  MoveL 1298 to (-37.11, 208.63, 290) mm, rotated rx -90 ry -25 rz 8.11 deg; joints [2.992, -45.692, 98.056, 40.659, -108.852, -6.827, -2568.107]
  MoveL 1299 to (-37.11, 208.63, 290) mm, rotated rx -90 ry -25 rz 8.11 deg; joints [2.992, -45.692, 98.056, 40.659, -108.852, -6.827, -2568.107]
  Set speed (60.0 mm/s)
  MoveL 1300 to (-43.85, 188.95, 290) mm, rotated rx -90 ry -25 rz 14.31 deg; joints [2.992, -46.574, 97.966, 40.447, -108.114, -7.494, -2574.314]
  Set speed (1000.0 mm/s)
  MoveL 1301 to (-43.85, 188.95, 290) mm, rotated rx -90 ry -25 rz 14.31 deg; joints [2.992, -46.574, 97.966, 40.447, -108.114, -7.494, -2574.314]
  Set speed (1000.0 mm/s)
  MoveL 1302 to (20.49, 309.71, 0) mm, rotated rx -90 ry -25 rz -148.94 deg; joints [-7.468, -50.346, 106.416, 34.531, -108.048, 0.653, -2411.057]
  MoveL 1303 to (20.49, 309.71, 0) mm, rotated rx -90 ry -25 rz -148.94 deg; joints [-7.468, -50.346, 106.416, 34.531, -108.048, 0.653, -2411.057]
  Set speed (60.0 mm/s)
  MoveL 1304 to (20.57, 330.51, 0) mm, rotated rx -90 ry -25 rz -144.34 deg; joints [-7.468, -51.311, 106.31, 34.338, -107.164, 0.017, -2415.665]
  Set speed (1000.0 mm/s)
  MoveL 1305 to (20.57, 330.51, 0) mm, rotated rx -90 ry -25 rz -144.34 deg; joints [-7.468, -51.311, 106.31, 34.338, -107.164, 0.017, -2415.665]
  Set speed (1000.0 mm/s)
  MoveL 1306 to (20.49, 309.71, 0) mm, rotated rx -90 ry -25 rz -148.94 deg; joints [-7.468, -50.346, 106.416, 34.531, -108.048, 0.653, -2411.057]
  MoveL 1307 to (20.49, 309.71, 0) mm, rotated rx -90 ry -25 rz -148.94 deg; joints [-7.468, -50.346, 106.416, 34.531, -108.048, 0.653, -2411.057]
  Set speed (60.0 mm/s)
  MoveL 1308 to (16.38, 311.06, 10) mm, rotated rx -90 ry -25 rz -145.01 deg; joints [-7.088, -50.246, 106.214, 34.77, -108.084, 0.408, -2414.985]
  MoveL 1309 to (11.76, 312.2, 20) mm, rotated rx -90 ry -25 rz -140.7 deg; joints [-6.709, -50.143, 106.006, 35.007, -108.12, 0.162, -2419.296]
  MoveL 1310 to (6.67, 313.01, 30) mm, rotated rx -90 ry -25 rz -136.04 deg; joints [-6.332, -50.036, 105.793, 35.242, -108.155, -0.085, -2423.955]
  MoveL 1311 to (1.18, 313.37, 40) mm, rotated rx -90 ry -25 rz -131.07 deg; joints [-5.956, -49.924, 105.573, 35.476, -108.19, -0.333, -2428.933]
  MoveL 1312 to (-4.64, 313.2, 50) mm, rotated rx -90 ry -25 rz -125.8 deg; joints [-5.581, -49.807, 105.347, 35.708, -108.224, -0.581, -2434.198]
  MoveL 1313 to (-10.69, 312.41, 60) mm, rotated rx -90 ry -25 rz -120.28 deg; joints [-5.207, -49.684, 105.115, 35.938, -108.259, -0.83, -2439.72]
  MoveL 1314 to (-16.86, 310.92, 70) mm, rotated rx -90 ry -25 rz -114.53 deg; joints [-4.834, -49.556, 104.876, 36.166, -108.295, -1.078, -2445.47]
  MoveL 1315 to (-23.03, 308.7, 80) mm, rotated rx -90 ry -25 rz -108.58 deg; joints [-4.463, -49.423, 104.632, 36.393, -108.331, -1.327, -2451.421]
  MoveL 1316 to (-29.06, 305.72, 90) mm, rotated rx -90 ry -25 rz -102.46 deg; joints [-4.093, -49.283, 104.382, 36.619, -108.368, -1.575, -2457.545]
  MoveL 1317 to (-34.83, 302, 100) mm, rotated rx -90 ry -25 rz -96.19 deg; joints [-3.725, -49.138, 104.126, 36.842, -108.405, -1.823, -2463.814]
  MoveL 1318 to (-40.19, 297.56, 110) mm, rotated rx -90 ry -25 rz -89.8 deg; joints [-3.358, -48.988, 103.864, 37.064, -108.442, -2.072, -2470.201]
  MoveL 1319 to (-45.04, 292.47, 120) mm, rotated rx -90 ry -25 rz -83.32 deg; joints [-2.992, -48.832, 103.595, 37.285, -108.48, -2.32, -2476.68]
  MoveL 1320 to (-49.26, 286.82, 130) mm, rotated rx -90 ry -25 rz -76.78 deg; joints [-2.628, -48.671, 103.321, 37.503, -108.518, -2.569, -2483.221]
  MoveL 1321 to (-52.77, 280.72, 140) mm, rotated rx -90 ry -25 rz -70.2 deg; joints [-2.265, -48.505, 103.04, 37.719, -108.556, -2.819, -2489.796]
  MoveL 1322 to (-55.51, 274.28, 150) mm, rotated rx -90 ry -25 rz -63.63 deg; joints [-1.904, -48.334, 102.753, 37.934, -108.592, -3.069, -2496.375]
  MoveL 1323 to (-57.45, 267.65, 160) mm, rotated rx -90 ry -25 rz -57.07 deg; joints [-1.544, -48.16, 102.46, 38.146, -108.628, -3.32, -2502.926]
  MoveL 1324 to (-58.59, 260.95, 170) mm, rotated rx -90 ry -25 rz -50.58 deg; joints [-1.185, -47.982, 102.161, 38.356, -108.662, -3.573, -2509.416]
  MoveL 1325 to (-58.95, 254.32, 180) mm, rotated rx -90 ry -25 rz -44.19 deg; joints [-0.828, -47.801, 101.855, 38.563, -108.694, -3.828, -2515.809]
  MoveL 1326 to (-58.59, 247.88, 190) mm, rotated rx -90 ry -25 rz -37.93 deg; joints [-0.473, -47.618, 101.543, 38.768, -108.724, -4.086, -2522.068]
  MoveL 1327 to (-57.57, 241.75, 200) mm, rotated rx -90 ry -25 rz -31.84 deg; joints [-0.119, -47.432, 101.224, 38.971, -108.752, -4.345, -2528.155]
  MoveL 1328 to (-56, 236.01, 210) mm, rotated rx -90 ry -25 rz -25.97 deg; joints [0.233, -47.244, 100.899, 39.17, -108.776, -4.608, -2534.028]
  MoveL 1329 to (-53.98, 230.73, 220) mm, rotated rx -90 ry -25 rz -20.35 deg; joints [0.584, -47.055, 100.567, 39.367, -108.797, -4.873, -2539.646]
  MoveL 1330 to (-51.62, 225.97, 230) mm, rotated rx -90 ry -25 rz -15.04 deg; joints [0.933, -46.864, 100.228, 39.56, -108.815, -5.142, -2544.964]
  MoveL 1331 to (-49.06, 221.75, 240) mm, rotated rx -90 ry -25 rz -10.06 deg; joints [1.28, -46.672, 99.883, 39.751, -108.83, -5.414, -2549.94]
  MoveL 1332 to (-46.4, 218.08, 250) mm, rotated rx -90 ry -25 rz -5.47 deg; joints [1.626, -46.479, 99.531, 39.939, -108.841, -5.69, -2554.527]
  MoveL 1333 to (-43.78, 214.95, 260) mm, rotated rx -90 ry -25 rz -1.32 deg; joints [1.97, -46.284, 99.173, 40.123, -108.849, -5.969, -2558.681]
  MoveL 1334 to (-41.29, 212.35, 270) mm, rotated rx -90 ry -25 rz 2.36 deg; joints [2.312, -46.089, 98.807, 40.305, -108.853, -6.252, -2562.358]
  MoveL 1335 to (-39.03, 210.26, 280) mm, rotated rx -90 ry -25 rz 5.51 deg; joints [2.653, -45.891, 98.435, 40.483, -108.854, -6.538, -2565.515]
  MoveL 1336 to (-37.11, 208.63, 290) mm, rotated rx -90 ry -25 rz 8.11 deg; joints [2.992, -45.692, 98.056, 40.659, -108.852, -6.827, -2568.107]
  Set speed (1000.0 mm/s)
  MoveL 1337 to (-37.11, 208.63, 290) mm, rotated rx -90 ry -25 rz 8.11 deg; joints [2.992, -45.692, 98.056, 40.659, -108.852, -6.827, -2568.107]
  Set speed (1000.0 mm/s)
  MoveL 1338 to (-43.85, 188.95, 290) mm, rotated rx -90 ry -25 rz 14.31 deg; joints [2.992, -46.574, 97.966, 40.447, -108.114, -7.494, -2574.314]
  MoveL 1339 to (-43.85, 188.95, 290) mm, rotated rx -90 ry -25 rz 14.31 deg; joints [2.992, -46.574, 97.966, 40.447, -108.114, -7.494, -2574.314]
  Set speed (60.0 mm/s)
  MoveL 1340 to (-46.6, 190.89, 280) mm, rotated rx -90 ry -25 rz 11.75 deg; joints [2.653, -46.775, 98.344, 40.272, -108.112, -7.203, -2571.748]
  MoveL 1341 to (-49.86, 193.4, 270) mm, rotated rx -90 ry -25 rz 8.62 deg; joints [2.312, -46.974, 98.716, 40.094, -108.107, -6.916, -2568.621]
  MoveL 1342 to (-53.49, 196.56, 260) mm, rotated rx -90 ry -25 rz 4.97 deg; joints [1.97, -47.172, 99.081, 39.913, -108.099, -6.633, -2564.974]
  MoveL 1343 to (-57.36, 200.4, 250) mm, rotated rx -90 ry -25 rz 0.85 deg; joints [1.626, -47.368, 99.44, 39.729, -108.088, -6.352, -2560.848]
  MoveL 1344 to (-61.34, 204.96, 240) mm, rotated rx -90 ry -25 rz -3.71 deg; joints [1.28, -47.563, 99.791, 39.542, -108.074, -6.075, -2556.286]
  MoveL 1345 to (-65.27, 210.27, 230) mm, rotated rx -90 ry -25 rz -8.67 deg; joints [0.933, -47.757, 100.136, 39.352, -108.055, -5.802, -2551.328]
  MoveL 1346 to (-68.98, 216.33, 220) mm, rotated rx -90 ry -25 rz -13.98 deg; joints [0.584, -47.949, 100.474, 39.159, -108.034, -5.532, -2546.018]
  MoveL 1347 to (-72.31, 223.11, 210) mm, rotated rx -90 ry -25 rz -19.6 deg; joints [0.233, -48.14, 100.805, 38.963, -108.008, -5.265, -2540.399]
  MoveL 1348 to (-75.1, 230.56, 200) mm, rotated rx -90 ry -25 rz -25.49 deg; joints [-0.119, -48.329, 101.13, 38.764, -107.98, -5.001, -2534.511]
  MoveL 1349 to (-77.2, 238.6, 190) mm, rotated rx -90 ry -25 rz -31.6 deg; joints [-0.473, -48.517, 101.448, 38.563, -107.948, -4.74, -2528.397]
  MoveL 1350 to (-78.47, 247.13, 180) mm, rotated rx -90 ry -25 rz -37.9 deg; joints [-0.828, -48.703, 101.76, 38.358, -107.914, -4.481, -2522.096]
  MoveL 1351 to (-78.79, 256, 170) mm, rotated rx -90 ry -25 rz -44.35 deg; joints [-1.185, -48.886, 102.065, 38.152, -107.877, -4.226, -2515.648]
  MoveL 1352 to (-78.09, 265.05, 160) mm, rotated rx -90 ry -25 rz -50.91 deg; joints [-1.544, -49.066, 102.363, 37.942, -107.838, -3.972, -2509.09]
  MoveL 1353 to (-76.31, 274.12, 150) mm, rotated rx -90 ry -25 rz -57.54 deg; joints [-1.904, -49.244, 102.656, 37.731, -107.797, -3.719, -2502.46]
  MoveL 1354 to (-73.44, 283.02, 140) mm, rotated rx -90 ry -25 rz -64.21 deg; joints [-2.265, -49.417, 102.942, 37.517, -107.754, -3.468, -2495.79]
  MoveL 1355 to (-69.5, 291.57, 130) mm, rotated rx -90 ry -25 rz -70.88 deg; joints [-2.628, -49.587, 103.221, 37.301, -107.711, -3.218, -2489.115]
  MoveL 1356 to (-64.57, 299.61, 120) mm, rotated rx -90 ry -25 rz -77.53 deg; joints [-2.992, -49.751, 103.495, 37.083, -107.667, -2.969, -2482.468]
  MoveL 1357 to (-58.74, 306.97, 110) mm, rotated rx -90 ry -25 rz -84.12 deg; joints [-3.358, -49.911, 103.762, 36.864, -107.624, -2.72, -2475.878]
  MoveL 1358 to (-52.14, 313.53, 100) mm, rotated rx -90 ry -25 rz -90.62 deg; joints [-3.725, -50.066, 104.024, 36.642, -107.58, -2.471, -2469.376]
  MoveL 1359 to (-44.91, 319.19, 90) mm, rotated rx -90 ry -25 rz -97.01 deg; joints [-4.093, -50.215, 104.279, 36.419, -107.536, -2.222, -2462.991]
  MoveL 1360 to (-37.24, 323.88, 80) mm, rotated rx -90 ry -25 rz -103.25 deg; joints [-4.463, -50.358, 104.529, 36.195, -107.494, -1.973, -2456.752]
  MoveL 1361 to (-29.3, 327.59, 70) mm, rotated rx -90 ry -25 rz -109.31 deg; joints [-4.834, -50.496, 104.772, 35.968, -107.451, -1.724, -2450.689]
  MoveL 1362 to (-21.27, 330.31, 60) mm, rotated rx -90 ry -25 rz -115.17 deg; joints [-5.207, -50.628, 105.01, 35.74, -107.41, -1.474, -2444.831]
  MoveL 1363 to (-13.31, 332.11, 50) mm, rotated rx -90 ry -25 rz -120.79 deg; joints [-5.581, -50.755, 105.242, 35.511, -107.369, -1.225, -2439.206]
  MoveL 1364 to (-5.58, 333.04, 40) mm, rotated rx -90 ry -25 rz -126.15 deg; joints [-5.956, -50.876, 105.467, 35.28, -107.328, -0.976, -2433.845]
  MoveL 1365 to (1.77, 333.22, 30) mm, rotated rx -90 ry -25 rz -131.22 deg; joints [-6.332, -50.991, 105.687, 35.047, -107.287, -0.727, -2428.779]
  MoveL 1366 to (8.64, 332.76, 20) mm, rotated rx -90 ry -25 rz -135.96 deg; joints [-6.709, -51.103, 105.901, 34.813, -107.247, -0.478, -2424.039]
  MoveL 1367 to (14.93, 331.81, 10) mm, rotated rx -90 ry -25 rz -140.34 deg; joints [-7.088, -51.209, 106.109, 34.576, -107.206, -0.23, -2419.656]
  MoveL 1368 to (20.57, 330.51, 0) mm, rotated rx -90 ry -25 rz -144.34 deg; joints [-7.468, -51.311, 106.31, 34.338, -107.164, 0.017, -2415.665]
  Set speed (1000.0 mm/s)
  MoveL 1369 to (20.57, 330.51, 0) mm, rotated rx -90 ry -25 rz -144.34 deg; joints [-7.468, -51.311, 106.31, 34.338, -107.164, 0.017, -2415.665]
  Set speed (1000.0 mm/s)
  MoveL 1370 to (-43.85, 188.95, 290) mm, rotated rx -90 ry -25 rz 14.31 deg; joints [2.992, -46.574, 97.966, 40.447, -108.114, -7.494, -2574.314]
  MoveL 1371 to (-43.85, 188.95, 290) mm, rotated rx -90 ry -25 rz 14.31 deg; joints [2.992, -46.574, 97.966, 40.447, -108.114, -7.494, -2574.314]
  Set speed (60.0 mm/s)
  MoveL 1372 to (-28.22, 202.67, 290) mm, rotated rx -90 ry -25 rz 19.2 deg; joints [2.992, -45.67, 98.058, 40.664, -108.87, -6.811, -2579.196]
  Set speed (1000.0 mm/s)
  MoveL 1373 to (-28.22, 202.67, 290) mm, rotated rx -90 ry -25 rz 19.2 deg; joints [2.992, -45.67, 98.058, 40.664, -108.87, -6.811, -2579.196]
  Set speed (1000.0 mm/s)
  MoveL 1374 to (20.57, 330.51, 0) mm, rotated rx -90 ry -25 rz -144.34 deg; joints [-7.468, -51.311, 106.31, 34.338, -107.164, 0.017, -2415.665]
  MoveL 1375 to (20.57, 330.51, 0) mm, rotated rx -90 ry -25 rz -144.34 deg; joints [-7.468, -51.311, 106.31, 34.338, -107.164, 0.017, -2415.665]
  Set speed (60.0 mm/s)
  MoveL 1376 to (10.16, 312.5, 0) mm, rotated rx -90 ry -25 rz -139.23 deg; joints [-7.468, -50.355, 106.415, 34.529, -108.039, 0.646, -2420.767]
  Set speed (1000.0 mm/s)
  MoveL 1377 to (10.16, 312.5, 0) mm, rotated rx -90 ry -25 rz -139.23 deg; joints [-7.468, -50.355, 106.415, 34.529, -108.039, 0.646, -2420.767]
  Set speed (1000.0 mm/s)
  MoveL 1378 to (20.57, 330.51, 0) mm, rotated rx -90 ry -25 rz -144.34 deg; joints [-7.468, -51.311, 106.31, 34.338, -107.164, 0.017, -2415.665]
  MoveL 1379 to (20.57, 330.51, 0) mm, rotated rx -90 ry -25 rz -144.34 deg; joints [-7.468, -51.311, 106.31, 34.338, -107.164, 0.017, -2415.665]
  Set speed (60.0 mm/s)
  MoveL 1380 to (14.93, 331.81, 10) mm, rotated rx -90 ry -25 rz -140.34 deg; joints [-7.088, -51.209, 106.109, 34.576, -107.206, -0.23, -2419.656]
  MoveL 1381 to (8.64, 332.76, 20) mm, rotated rx -90 ry -25 rz -135.96 deg; joints [-6.709, -51.103, 105.901, 34.813, -107.247, -0.478, -2424.039]
  MoveL 1382 to (1.77, 333.22, 30) mm, rotated rx -90 ry -25 rz -131.22 deg; joints [-6.332, -50.991, 105.687, 35.047, -107.287, -0.727, -2428.779]
  MoveL 1383 to (-5.58, 333.04, 40) mm, rotated rx -90 ry -25 rz -126.15 deg; joints [-5.956, -50.876, 105.467, 35.28, -107.328, -0.976, -2433.845]
  MoveL 1384 to (-13.31, 332.11, 50) mm, rotated rx -90 ry -25 rz -120.79 deg; joints [-5.581, -50.755, 105.242, 35.511, -107.369, -1.225, -2439.206]
  MoveL 1385 to (-21.27, 330.31, 60) mm, rotated rx -90 ry -25 rz -115.17 deg; joints [-5.207, -50.628, 105.01, 35.74, -107.41, -1.474, -2444.831]
  MoveL 1386 to (-29.3, 327.59, 70) mm, rotated rx -90 ry -25 rz -109.31 deg; joints [-4.834, -50.496, 104.772, 35.968, -107.451, -1.724, -2450.689]
  MoveL 1387 to (-37.24, 323.88, 80) mm, rotated rx -90 ry -25 rz -103.25 deg; joints [-4.463, -50.358, 104.529, 36.195, -107.494, -1.973, -2456.752]
  MoveL 1388 to (-44.91, 319.19, 90) mm, rotated rx -90 ry -25 rz -97.01 deg; joints [-4.093, -50.215, 104.279, 36.419, -107.536, -2.222, -2462.991]
  MoveL 1389 to (-52.14, 313.53, 100) mm, rotated rx -90 ry -25 rz -90.62 deg; joints [-3.725, -50.066, 104.024, 36.642, -107.58, -2.471, -2469.376]
  MoveL 1390 to (-58.74, 306.97, 110) mm, rotated rx -90 ry -25 rz -84.12 deg; joints [-3.358, -49.911, 103.762, 36.864, -107.624, -2.72, -2475.878]
  MoveL 1391 to (-64.57, 299.61, 120) mm, rotated rx -90 ry -25 rz -77.53 deg; joints [-2.992, -49.751, 103.495, 37.083, -107.667, -2.969, -2482.468]
  MoveL 1392 to (-69.5, 291.57, 130) mm, rotated rx -90 ry -25 rz -70.88 deg; joints [-2.628, -49.587, 103.221, 37.301, -107.711, -3.218, -2489.115]
  MoveL 1393 to (-73.44, 283.02, 140) mm, rotated rx -90 ry -25 rz -64.21 deg; joints [-2.265, -49.417, 102.942, 37.517, -107.754, -3.468, -2495.79]
  MoveL 1394 to (-76.31, 274.12, 150) mm, rotated rx -90 ry -25 rz -57.54 deg; joints [-1.904, -49.244, 102.656, 37.731, -107.797, -3.719, -2502.46]
  MoveL 1395 to (-78.09, 265.05, 160) mm, rotated rx -90 ry -25 rz -50.91 deg; joints [-1.544, -49.066, 102.363, 37.942, -107.838, -3.972, -2509.09]
  MoveL 1396 to (-78.79, 256, 170) mm, rotated rx -90 ry -25 rz -44.35 deg; joints [-1.185, -48.886, 102.065, 38.152, -107.877, -4.226, -2515.648]
  MoveL 1397 to (-78.47, 247.13, 180) mm, rotated rx -90 ry -25 rz -37.9 deg; joints [-0.828, -48.703, 101.76, 38.358, -107.914, -4.481, -2522.096]
  MoveL 1398 to (-77.2, 238.6, 190) mm, rotated rx -90 ry -25 rz -31.6 deg; joints [-0.473, -48.517, 101.448, 38.563, -107.948, -4.74, -2528.397]
  MoveL 1399 to (-75.1, 230.56, 200) mm, rotated rx -90 ry -25 rz -25.49 deg; joints [-0.119, -48.329, 101.13, 38.764, -107.98, -5.001, -2534.511]
  MoveL 1400 to (-72.31, 223.11, 210) mm, rotated rx -90 ry -25 rz -19.6 deg; joints [0.233, -48.14, 100.805, 38.963, -108.008, -5.265, -2540.399]
  MoveL 1401 to (-68.98, 216.33, 220) mm, rotated rx -90 ry -25 rz -13.98 deg; joints [0.584, -47.949, 100.474, 39.159, -108.034, -5.532, -2546.018]
  MoveL 1402 to (-65.27, 210.27, 230) mm, rotated rx -90 ry -25 rz -8.67 deg; joints [0.933, -47.757, 100.136, 39.352, -108.055, -5.802, -2551.328]
  MoveL 1403 to (-61.34, 204.96, 240) mm, rotated rx -90 ry -25 rz -3.71 deg; joints [1.28, -47.563, 99.791, 39.542, -108.074, -6.075, -2556.286]
  MoveL 1404 to (-57.36, 200.4, 250) mm, rotated rx -90 ry -25 rz 0.85 deg; joints [1.626, -47.368, 99.44, 39.729, -108.088, -6.352, -2560.848]
  MoveL 1405 to (-53.49, 196.56, 260) mm, rotated rx -90 ry -25 rz 4.97 deg; joints [1.97, -47.172, 99.081, 39.913, -108.099, -6.633, -2564.974]
  MoveL 1406 to (-49.86, 193.4, 270) mm, rotated rx -90 ry -25 rz 8.62 deg; joints [2.312, -46.974, 98.716, 40.094, -108.107, -6.916, -2568.621]
  MoveL 1407 to (-46.6, 190.89, 280) mm, rotated rx -90 ry -25 rz 11.75 deg; joints [2.653, -46.775, 98.344, 40.272, -108.112, -7.203, -2571.748]
  MoveL 1408 to (-43.85, 188.95, 290) mm, rotated rx -90 ry -25 rz 14.31 deg; joints [2.992, -46.574, 97.966, 40.447, -108.114, -7.494, -2574.314]
  Set speed (1000.0 mm/s)
  MoveL 1409 to (-43.85, 188.95, 290) mm, rotated rx -90 ry -25 rz 14.31 deg; joints [2.992, -46.574, 97.966, 40.447, -108.114, -7.494, -2574.314]
  Set speed (1000.0 mm/s)
  MoveL 1410 to (-28.22, 202.67, 290) mm, rotated rx -90 ry -25 rz 19.2 deg; joints [2.992, -45.67, 98.058, 40.664, -108.87, -6.811, -2579.196]
  MoveL 1411 to (-28.22, 202.67, 290) mm, rotated rx -90 ry -25 rz 19.2 deg; joints [2.992, -45.67, 98.058, 40.664, -108.87, -6.811, -2579.196]
  Set speed (60.0 mm/s)
  MoveL 1412 to (-30.4, 203.93, 280) mm, rotated rx -90 ry -25 rz 16.58 deg; joints [2.653, -45.868, 98.437, 40.489, -108.873, -6.521, -2576.579]
  MoveL 1413 to (-33, 205.58, 270) mm, rotated rx -90 ry -25 rz 13.39 deg; joints [2.312, -46.064, 98.809, 40.311, -108.874, -6.234, -2573.391]
  MoveL 1414 to (-35.92, 207.69, 260) mm, rotated rx -90 ry -25 rz 9.67 deg; joints [1.97, -46.258, 99.175, 40.13, -108.871, -5.95, -2569.674]
  MoveL 1415 to (-39.07, 210.28, 250) mm, rotated rx -90 ry -25 rz 5.47 deg; joints [1.626, -46.451, 99.533, 39.946, -108.865, -5.669, -2565.473]
  MoveL 1416 to (-42.34, 213.41, 240) mm, rotated rx -90 ry -25 rz 0.83 deg; joints [1.28, -46.642, 99.885, 39.758, -108.855, -5.392, -2560.831]
  MoveL 1417 to (-45.62, 217.1, 230) mm, rotated rx -90 ry -25 rz -4.21 deg; joints [0.933, -46.832, 100.231, 39.568, -108.842, -5.119, -2555.794]
  MoveL 1418 to (-48.8, 221.36, 220) mm, rotated rx -90 ry -25 rz -9.59 deg; joints [0.584, -47.021, 100.57, 39.375, -108.826, -4.849, -2550.406]
  MoveL 1419 to (-51.74, 226.19, 210) mm, rotated rx -90 ry -25 rz -15.29 deg; joints [0.233, -47.209, 100.902, 39.178, -108.806, -4.582, -2544.713]
  MoveL 1420 to (-54.33, 231.55, 200) mm, rotated rx -90 ry -25 rz -21.24 deg; joints [-0.119, -47.395, 101.227, 38.979, -108.783, -4.319, -2538.758]
  MoveL 1421 to (-56.44, 237.4, 190) mm, rotated rx -90 ry -25 rz -27.41 deg; joints [-0.473, -47.58, 101.546, 38.777, -108.756, -4.059, -2532.587]
  MoveL 1422 to (-57.96, 243.66, 180) mm, rotated rx -90 ry -25 rz -33.76 deg; joints [-0.828, -47.763, 101.858, 38.572, -108.727, -3.801, -2526.24]
  MoveL 1423 to (-58.8, 250.25, 170) mm, rotated rx -90 ry -25 rz -40.24 deg; joints [-1.185, -47.944, 102.164, 38.365, -108.694, -3.547, -2519.76]
  MoveL 1424 to (-58.89, 257.04, 160) mm, rotated rx -90 ry -25 rz -46.82 deg; joints [-1.544, -48.123, 102.464, 38.154, -108.66, -3.294, -2513.183]
  MoveL 1425 to (-58.18, 263.92, 150) mm, rotated rx -90 ry -25 rz -53.45 deg; joints [-1.904, -48.298, 102.757, 37.942, -108.623, -3.043, -2506.549]
  MoveL 1426 to (-56.65, 270.74, 140) mm, rotated rx -90 ry -25 rz -60.11 deg; joints [-2.265, -48.47, 103.043, 37.727, -108.585, -2.794, -2499.89]
  MoveL 1427 to (-54.3, 277.38, 130) mm, rotated rx -90 ry -25 rz -66.76 deg; joints [-2.628, -48.638, 103.324, 37.51, -108.546, -2.546, -2493.241]
  MoveL 1428 to (-51.17, 283.7, 120) mm, rotated rx -90 ry -25 rz -73.37 deg; joints [-2.992, -48.802, 103.598, 37.291, -108.506, -2.299, -2486.632]
  MoveL 1429 to (-47.33, 289.58, 110) mm, rotated rx -90 ry -25 rz -79.91 deg; joints [-3.358, -48.961, 103.866, 37.07, -108.466, -2.053, -2480.094]
  MoveL 1430 to (-42.85, 294.92, 100) mm, rotated rx -90 ry -25 rz -86.35 deg; joints [-3.725, -49.114, 104.128, 36.848, -108.426, -1.807, -2473.654]
  MoveL 1431 to (-37.86, 299.62, 90) mm, rotated rx -90 ry -25 rz -92.66 deg; joints [-4.093, -49.263, 104.384, 36.623, -108.386, -1.561, -2467.341]
  MoveL 1432 to (-32.46, 303.64, 80) mm, rotated rx -90 ry -25 rz -98.82 deg; joints [-4.463, -49.406, 104.634, 36.397, -108.346, -1.315, -2461.181]
  MoveL 1433 to (-26.8, 306.94, 70) mm, rotated rx -90 ry -25 rz -104.8 deg; joints [-4.834, -49.543, 104.878, 36.169, -108.307, -1.069, -2455.202]
  MoveL 1434 to (-21, 309.52, 60) mm, rotated rx -90 ry -25 rz -110.57 deg; joints [-5.207, -49.675, 105.115, 35.94, -108.268, -0.823, -2449.431]
  MoveL 1435 to (-15.19, 311.39, 50) mm, rotated rx -90 ry -25 rz -116.1 deg; joints [-5.581, -49.801, 105.347, 35.709, -108.23, -0.577, -2443.896]
  MoveL 1436 to (-9.5, 312.61, 40) mm, rotated rx -90 ry -25 rz -121.38 deg; joints [-5.956, -49.921, 105.573, 35.476, -108.192, -0.331, -2438.624]
  MoveL 1437 to (-4.03, 313.25, 30) mm, rotated rx -90 ry -25 rz -126.35 deg; joints [-6.332, -50.037, 105.793, 35.242, -108.154, -0.086, -2433.645]
  MoveL 1438 to (1.12, 313.37, 20) mm, rotated rx -90 ry -25 rz -131.01 deg; joints [-6.709, -50.147, 106.006, 35.006, -108.116, 0.159, -2428.989]
  MoveL 1439 to (5.87, 313.09, 10) mm, rotated rx -90 ry -25 rz -135.31 deg; joints [-7.088, -50.253, 106.214, 34.768, -108.078, 0.403, -2424.685]
  MoveL 1440 to (10.16, 312.5, 0) mm, rotated rx -90 ry -25 rz -139.23 deg; joints [-7.468, -50.355, 106.415, 34.529, -108.039, 0.646, -2420.767]
  Set speed (1000.0 mm/s)
  MoveL 1441 to (10.16, 312.5, 0) mm, rotated rx -90 ry -25 rz -139.23 deg; joints [-7.468, -50.355, 106.415, 34.529, -108.039, 0.646, -2420.767]
